TYPE "MotorSts"
VERSION : 0.1
// Block: MotorSts
   STRUCT
      AlarmPresence : Bool;
      RunPermitted : Bool;
      Running : Bool;
   END_STRUCT;

END_TYPE
